TYPE ST_Parameter :
STRUCT
END_STRUCT
END_TYPE

(* stored: Version 1.1.0.1, ProductVersion 3.1.4024.10
   DUT ST_Parameter: Id {e93b63fb-60cf-4270-a281-be4bce1daaeb} *)
